% RSLogix 500 project PLC Level 2 Project 1.RSS, saved by version 8.30.00.16 %
PROJECT "UNTITLED"    % processor: Bul.1763 MicroLogix 1100 Series B %

PROGRAM FILES
  LAD 2 "MAIN"  3 rungs
  LAD 3 "DIG IO"  5 rungs
  LAD 5 "CTRL LOGIC"  9 rungs

DATA FILES
  O0 OUTPUT  4 elements
  I1 INPUT  6 elements
  S2 STATUS  66 elements
  B3 BINARY  1 elements
  T4 TIMER  3 elements
  C5 COUNTER  1 elements
  R6 CONTROL  1 elements
  N7 INTEGER  1 elements
  F8 FLOAT  1 elements

LADDER 2 "MAIN"
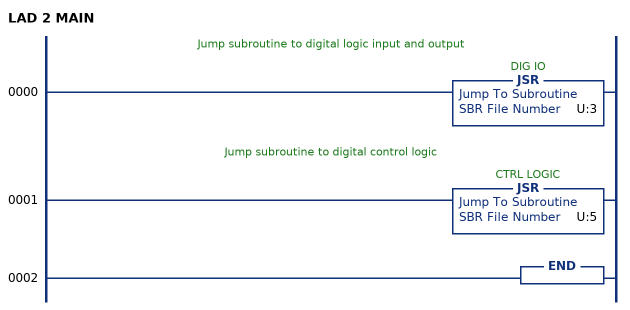
% Rung: 0 %
% Jump subroutine to digital logic input and output %
SOR JSR U:3 EOR
%   U:3  "DIG IO" %
% Rung: 1 %
% Jump subroutine to digital control logic %
SOR JSR U:5 EOR
%   U:5  "CTRL LOGIC" %
% Rung: 2 %
SOR END EOR

LADDER 3 "DIG IO"
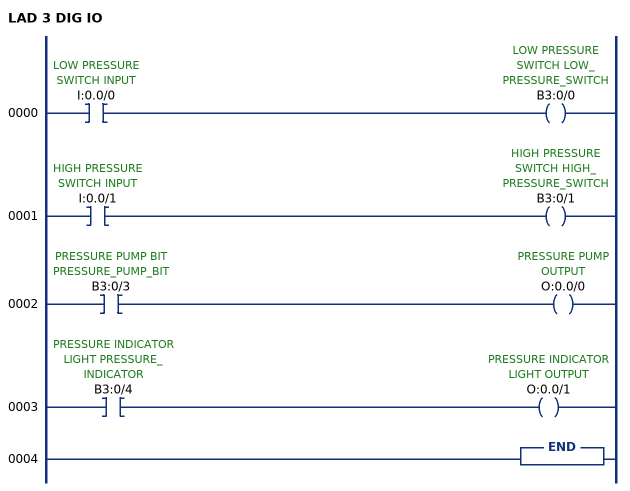
% Rung: 0 %
SOR XIC I:0.0/0 OTE B3:0/0 EOR
%   I:0.0/0  "LOW PRESSURE SWITCH INPUT" %
%   B3:0/0  LOW_PRESSURE_SWITCH  "LOW PRESSURE SWITCH" %
% Rung: 1 %
SOR XIC I:0.0/1 OTE B3:0/1 EOR
%   I:0.0/1  "HIGH PRESSURE SWITCH INPUT" %
%   B3:0/1  HIGH_PRESSURE_SWITCH  "HIGH PRESSURE SWITCH" %
% Rung: 2 %
SOR XIC B3:0/3 OTE O:0.0/0 EOR
%   B3:0/3  PRESSURE_PUMP_BIT  "PRESSURE PUMP BIT" %
%   O:0.0/0  "PRESSURE PUMP OUTPUT" %
% Rung: 3 %
SOR XIC B3:0/4 OTE O:0.0/1 EOR
%   B3:0/4  PRESSURE_INDICATOR  "PRESSURE INDICATOR LIGHT" %
%   O:0.0/1  "PRESSURE INDICATOR LIGHT OUTPUT" %
% Rung: 4 %
SOR END EOR

LADDER 5 "CTRL LOGIC"
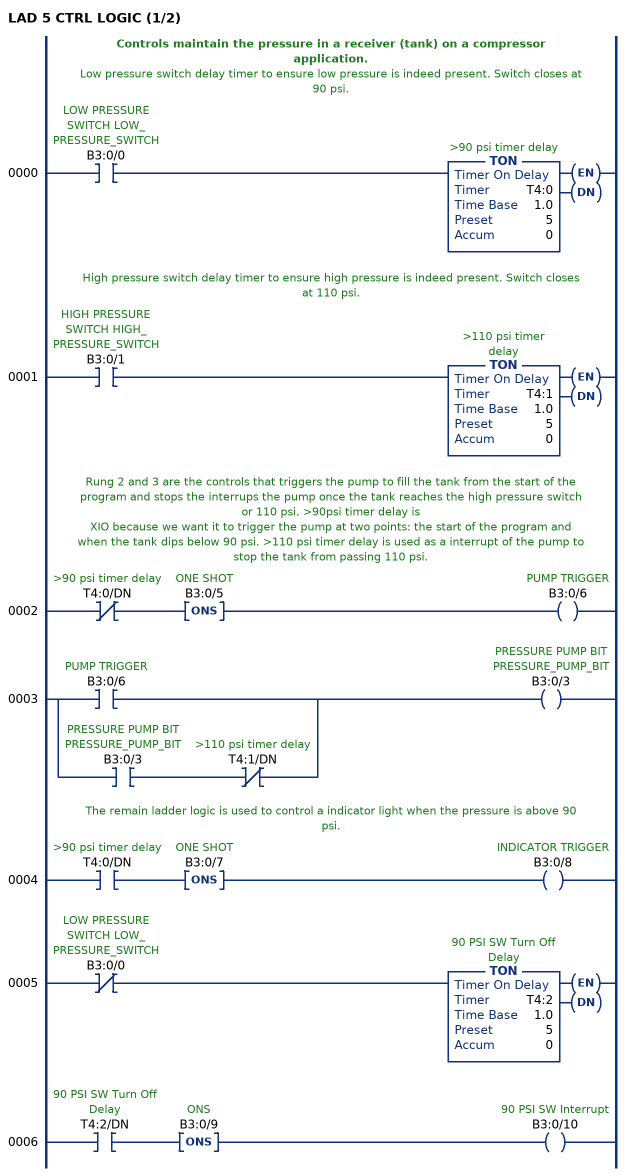
% Rung: 0 %
% TITLE: Controls maintain the pressure in a receiver (tank) on a compressor application. %
% Low pressure switch delay timer to ensure low pressure is indeed present. Switch closes at 90 psi. %
SOR XIC B3:0/0 TON T4:0 1.0 5 0 EOR
%   B3:0/0  LOW_PRESSURE_SWITCH  "LOW PRESSURE SWITCH" %
%   T4:0  ">90 psi timer delay" %
% Rung: 1 %
% High pressure switch delay timer to ensure high pressure is indeed present. Switch closes at 110 psi. %
SOR XIC B3:0/1 TON T4:1 1.0 5 0 EOR
%   B3:0/1  HIGH_PRESSURE_SWITCH  "HIGH PRESSURE SWITCH" %
%   T4:1  ">110 psi timer delay" %
% Rung: 2 %
%  Rung 2 and 3 are the controls that triggers the pump to fill the tank from the start of the program and stops the interrups the pump once the tank reaches the high pressure switch or 110 psi. >90psi timer delay is
% XIO because we want it to trigger the pump at two points: the start of the program and when the tank dips below 90 psi. >110 psi timer delay is used as a interrupt of the pump to stop the tank from passing 110 psi. %
SOR XIO T4:0/DN ONS B3:0/5 OTE B3:0/6 EOR
%   T4:0  ">90 psi timer delay" %
%   B3:0/5  "ONE SHOT" %
%   B3:0/6  "PUMP TRIGGER" %
% Rung: 3 %
SOR BST XIC B3:0/6 NXB XIC B3:0/3 XIO T4:1/DN BND OTE B3:0/3 EOR
%   B3:0/6  "PUMP TRIGGER" %
%   B3:0/3  PRESSURE_PUMP_BIT  "PRESSURE PUMP BIT" %
%   T4:1/DN  ">110 psi timer delay" %
% Rung: 4 %
% The remain ladder logic is used to control a indicator light when the pressure is above 90 psi. %
SOR XIC T4:0/DN ONS B3:0/7 OTE B3:0/8 EOR
%   T4:0  ">90 psi timer delay" %
%   B3:0/7  "ONE SHOT" %
%   B3:0/8  "INDICATOR TRIGGER" %
% Rung: 5 %
SOR XIO B3:0/0 TON T4:2 1.0 5 0 EOR
%   B3:0/0  LOW_PRESSURE_SWITCH  "LOW PRESSURE SWITCH" %
%   T4:2  "90 PSI SW Turn Off Delay" %
% Rung: 6 %
SOR XIC T4:2/DN ONS B3:0/9 OTE B3:0/10 EOR
%   T4:2  "90 PSI SW Turn Off Delay" %
%   B3:0/9  "ONS" %
%   B3:0/10  "90 PSI SW Interrupt" %

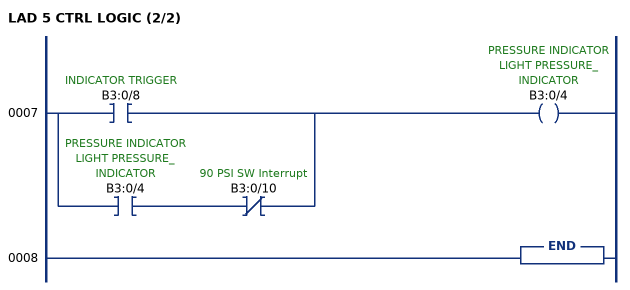
% Rung: 7 %
SOR BST XIC B3:0/8 NXB XIC B3:0/4 XIO B3:0/10 BND OTE B3:0/4 EOR
%   B3:0/8  "INDICATOR TRIGGER" %
%   B3:0/4  PRESSURE_INDICATOR  "PRESSURE INDICATOR LIGHT" %
%   B3:0/10  "90 PSI SW Interrupt" %
% Rung: 8 %
SOR END EOR

OTHER DOCUMENTED ADDRESSES
  T4:1/0  ">90 psi timer delay"
  U:4  "DIG OUT"
  U:6  "ALARMS"

DATA TABLE (non-zero values as saved)
DATA T4
% .PRE .ACC %
% T4:0 % 5 0
% T4:1 % 5 0
% T4:2 % 5 0
